INTERFACE I_Request EXTENDS I_Disposable

PROPERTY PUBLIC CreatedTimestamp : I_Timestamp
GET
END_GET
END_PROPERTY

PROPERTY PUBLIC Header : I_Header
GET
END_GET
END_PROPERTY

PROPERTY PUBLIC PayloadAddress : POINTER TO STRING
GET
END_GET
END_PROPERTY

PROPERTY PUBLIC PayloadSizeInBytes : UDINT
GET
END_GET
END_PROPERTY

END_INTERFACE

(* stored: Version 1.1.0.1, ProductVersion 3.1.4026.13
   Itf I_Request: Id {2caff5d7-2d1c-4288-ba94-1a88818d59b5}
   Property CreatedTimestamp: Id {366fc398-6ea4-4ff4-91de-75eeb259da0e}
   Get Get: Id {fa280de4-94ad-4c5e-b918-42ad21a2df4d}
   Property Header: Id {60487914-5942-4ffc-8f2b-5ab23e268ad3}
   Get Get: Id {8056231d-fc72-42f6-abaa-59858b85d4ac}
   Property PayloadAddress: Id {36a84d33-cc2a-4d0d-861e-47596faf4cda}
   Get Get: Id {f96c17f9-1572-461c-a2e5-15ee8a31d26b}
   Property PayloadSizeInBytes: Id {c597a2ed-0bf1-402d-8922-e727ddf7481b}
   Get Get: Id {bc9d3533-aac7-44a7-a73a-335762cc29df} *)
